{attribute 'GeneratedUsingTerminal: CU1124-0000-0016'}
{attribute addProperty BoxType "CU1124-0000-0016"}
{attribute addProperty Id "InfoDataAT %I*InfoData_6F19DB2B2"}
{attribute addProperty CRC "532711307"}
{attribute addProperty Size "2"}
TYPE CU1124_1FC0878B EXTENDS EtcSlaveTerminalBase_947E5A46 :
STRUCT
	{attribute addProperty Name "InfoData"}
	InfoData : InfoData_6F19DB2B;
END_STRUCT
END_TYPE

(* stored: Version 1.2.0.0, ProductVersion 3.1.4024.9
   DUT CU1124_1FC0878B: Id {dcab424b-d570-428b-af5e-70fb22fe5cb8} *)
